FUNCTION ImageHasElementType : BOOL
VAR_INPUT
	Image : ITcVnImage;
	ElementType : ETcVnElementType;
END_VAR

IF NOT IsValidImage(Image) THEN
	RETURN;
END_IF

ImageHasElementType := (ElementType = GetETcVnElementTypeFromImage(Image));

END_FUNCTION

(* stored: Version 1.1.0.1, ProductVersion 3.1.4024.13
   POU ImageHasElementType: Id {bc1fce88-dff5-48ea-b3c5-f51831dcb300}, SpecialFunc None *)
